PROGRAM PRG_CASE_DuplicateUpdateToDBManual
VAR
	fbCase_DuplicateUpdateToDB		: FB_CASE_DuplicateUpdateToDB;
	
	(* Data/Iterators for Init function/method *)
	rTrigDataInit			: R_TRIG;
	bDataInit				: BOOL;
	iOuter					: INT;
	iPack					: INT;
	sPackNum				: STRING;
	sOuterNum				: STRING;
	sPackCode				: STRING;
	stProductInstruction	: ST_PCM_Status;
	
	
	(* Inputs *)	
	bExecute						: BOOL;		(* set TRUE to archive OAC files *)
	bUseInterimCodeForValidation	: BOOL;
	
	
	(* In/Out *)
	aOCVPackStatus			: ARRAY[1..cMAX_OUTER_STATUS_QUEUE] OF ST_OUTER_Status;	(* Outer status array *)
	aOuterStatus			: ARRAY[1..cMAX_OUTER_STATUS_QUEUE] OF ST_OUTER_Status;	(* Outer status array *)
	
	stOCVDataDB							: ST_DB_OCVDataCtrl;
	stOACDataDB							: ST_DB_OACDataCtrl;
	
	stOuterBarcodeDuplicate				: ST_RejectItems;
	stOuterDuplicatedPackCodesFound		: ST_RejectItems;
	
	stCodeInfo_Pack				: ST_CodeInfo;
	stCodeInfo_Intermediate		: ST_CodeInfo;
	stCodeInfo_Outer			: ST_CodeInfo;
	
	stCACData					: ST_CAC_Data;
	
	(* Outputs *)
	bDone 					: BOOL;		(* TRUE = OAC archive complete *)
	bBusy 					: BOOL;		(* TRUE = OAC archive active *)
	bError 					: BOOL;		(* TRUE = OAC archive error *)
	nErrorID				: UDINT;	(* error code *)

	nOACFilesBlocked		: UINT;
	nOCVFilesBlocked		: UINT;
	stDaigOACDataDB			: ST_DB_OACDataCtrl;
	stDiagOCVDataDB			: ST_DB_OCVDataCtrl;
	
	
END_VAR

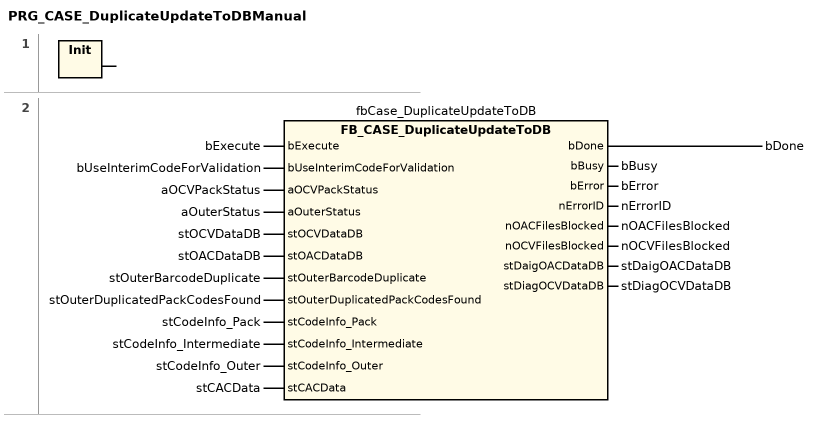
// NETWORK 1
Init();

// NETWORK 2
fbCase_DuplicateUpdateToDB(
    bExecute := bExecute,
    bUseInterimCodeForValidation := bUseInterimCodeForValidation,
    aOCVPackStatus := aOCVPackStatus,
    aOuterStatus := aOuterStatus,
    stOCVDataDB := stOCVDataDB,
    stOACDataDB := stOACDataDB,
    stOuterBarcodeDuplicate := stOuterBarcodeDuplicate,
    stOuterDuplicatedPackCodesFound := stOuterDuplicatedPackCodesFound,
    stCodeInfo_Pack := stCodeInfo_Pack,
    stCodeInfo_Intermediate := stCodeInfo_Intermediate,
    stCodeInfo_Outer := stCodeInfo_Outer,
    stCACData := stCACData,
    bBusy => bBusy,
    bError => bError,
    nErrorID => nErrorID,
    nOACFilesBlocked => nOACFilesBlocked,
    nOCVFilesBlocked => nOCVFilesBlocked,
    stDaigOACDataDB => stDaigOACDataDB,
    stDiagOCVDataDB => stDiagOCVDataDB); // FB_CASE_DuplicateUpdateToDB
bDone := fbCase_DuplicateUpdateToDB.bDone;

ACTION Init:

rTrigDataInit(CLK := bDataInit);

IF rTrigDataInit.Q THEN
	
	stProductInstruction.nOutersPerCase		:= 50;
	stProductInstruction.nPacksPerOuter 	:= 10;
	
	stCACData.NumberOfOuters	:= 50;
	

	FOR iOuter := 1 TO stProductInstruction.nOutersPerCase DO
		(* Ustaw outer *)
		stCACData.Outer[iOuter].Barcode    := CONCAT('OUTER', INT_TO_STRING(iOuter));
		stCACData.Outer[iOuter].OuterCodeStatus := 5;
		
		stCACData.Outer[iOuter].OuterRejectID	:= 0;
		
		
		FOR iPack := 1 TO stProductInstruction.nPacksPerOuter DO
			(* Pack number z zerami *)
			sPackNum := CONCAT('0', INT_TO_STRING(iPack));  (* dla 1-9: '01'-'09' *)
			IF iPack = 10 THEN
				sPackNum := '10';
			END_IF;
			
			(* Outer number z zerami dla 1-9 *)
			sOuterNum := CONCAT('0', INT_TO_STRING(iOuter));
			IF iOuter >= 10 THEN
				sOuterNum := INT_TO_STRING(iOuter);
			END_IF;
			
			(* Sklej pack code *)
			sPackCode := CONCAT(CONCAT('PACK', sPackNum), CONCAT('OUTER', sOuterNum));
			
			(* Przypisz *)
			stCACData.Outer[iOuter].PackCode[iPack]			:= sPackCode;
			stCACData.Outer[iOuter].PackCodeStatus[iPack]	:= 5;
			stCACData.Outer[iOuter].PackRejectID[iPack]		:= 0;
			
		END_FOR;
	END_FOR;	
	
END_IF
END_ACTION

END_PROGRAM

(* stored: Version 1.1.0.1
   POU PRG_CASE_DuplicateUpdateToDBManual: Id {6b38db0a-448f-4f87-8f93-153be185d66c}, SpecialFunc None
   Action Init: Id {ca01388e-369c-4012-9972-acc0938736d5} *)
